FUNCTION_BLOCK FB_MyProjectEvents EXTENDS FB_BA_ProjectEventSubscriber

METHOD PROTECTED OnProjectStateChanged
VAR_INPUT
	eState			: E_BA_ProjectState;
END_VAR
// Sample 1) Evaluate project state.
CASE (eState) OF
	E_BA_ProjectState.eFirstOpCycle:
		F_BA_LogMessage(ADSLOG_MSGTYPE_HINT, 'OPSC04', 'Initialization done: project is operational.');
	
	E_BA_ProjectState.Error:
		F_BA_LogMessage(ADSLOG_MSGTYPE_HINT, 'OPSC07', 'Initialization failed!');
	
END_CASE
END_METHOD

END_FUNCTION_BLOCK

(* stored: Version 1.1.0.1, ProductVersion 3.1.4024.12
   POU FB_MyProjectEvents: Id {4b156194-a872-4ef0-9daa-e7f0b809e2f4}, SpecialFunc None
   Folder [Protected] Events: Id {98751e3e-8e8c-4565-ad7f-46b621dbde9d}
   Method OnProjectStateChanged: Id {2b385d05-fa2e-4c3d-be6e-0f8478e619ac} *)
